
// =================================================================================
// Improved_Gluing_FC_SCL.scl
// Function: FC_Save_Current_Values_V6
// Version: 6.0 (FINAL)
//
// Description:
// FINAL version incorporating all user feedback.
// This function saves a snapshot of all live machine values into the final
// descriptive recipe structure, "UDT_ST10_Recipe_V3".
//
// - IAI axes are correctly mapped to the 3-axis gluing nozzle.
// - V90 axes are correctly mapped to their turntable/jig functions.
// - Does not use loops for positions; every parameter is saved explicitly.
//
// The source DBs ("Gluing_Nozzle_X_DB", "Ring_Table_1_DB", etc.) are placeholders
// and must be replaced with the actual DBs containing the live taught values.
// =================================================================================

FUNCTION "FC_Save_Current_Values_V6" : Void
{ S7_Optimized_Access := 'TRUE' }
VAR_TEMP
   // No loop variables needed
END_VAR

BEGIN
    // =================================================================================
    // 3-AXIS GLUING NOZZLE (IAI Axes)
    // =================================================================================
    "DB_ST10_Recipe".Motion.Gluing_Nozzle_X := "Gluing_Nozzle_X_DB".Live.Positions;
    "DB_ST10_Recipe".Motion.Gluing_Nozzle_Y := "Gluing_Nozzle_Y_DB".Live.Positions;
    "DB_ST10_Recipe".Motion.Gluing_Nozzle_Z := "Gluing_Nozzle_Z_DB".Live.Positions;

    // =================================================================================
    // ROTARY AXES (V90 Servos) - CORRECTED MAPPING
    // =================================================================================

    // --- V90 A1: Ring Turntable 1 ---
    "DB_ST10_Recipe".Motion.Ring_Turntable_Axis_1.Home              := "Ring_Table_1_DB".Live.Positions.Home;
    "DB_ST10_Recipe".Motion.Ring_Turntable_Axis_1.Load_Unload_Pos   := "Ring_Table_1_DB".Live.Positions.Load_Unload_Pos;
    "DB_ST10_Recipe".Motion.Ring_Turntable_Axis_1.Work_Pos_1        := "Ring_Table_1_DB".Live.Positions.Work_Pos_1;
    "DB_ST10_Recipe".Motion.Ring_Turntable_Axis_1.Work_Pos_2        := "Ring_Table_1_DB".Live.Positions.Work_Pos_2;
    // ...etc for spares

    // --- V90 A2: Shaft Scan Turntable ---
    "DB_ST10_Recipe".Motion.Shaft_Scan_Turntable_Axis.Home              := "Shaft_Scan_Table_DB".Live.Positions.Home;
    "DB_ST10_Recipe".Motion.Shaft_Scan_Turntable_Axis.Load_Unload_Pos   := "Shaft_Scan_Table_DB".Live.Positions.Load_Unload_Pos;
    "DB_ST10_Recipe".Motion.Shaft_Scan_Turntable_Axis.Work_Pos_1        := "Shaft_Scan_Table_DB".Live.Positions.Work_Pos_1;
    "DB_ST10_Recipe".Motion.Shaft_Scan_Turntable_Axis.Work_Pos_2        := "Shaft_Scan_Table_DB".Live.Positions.Work_Pos_2;
    // ...etc for spares

    // --- V90 A3: Gluing Rotary Jig ---
    "DB_ST10_Recipe".Motion.Gluing_Rotary_Jig_Axis.Home              := "Gluing_Jig_DB".Live.Positions.Home;
    "DB_ST10_Recipe".Motion.Gluing_Rotary_Jig_Axis.Load_Unload_Pos   := "Gluing_Jig_DB".Live.Positions.Load_Unload_Pos;
    "DB_ST10_Recipe".Motion.Gluing_Rotary_Jig_Axis.Work_Pos_1        := "Gluing_Jig_DB".Live.Positions.Work_Pos_1;
    "DB_ST10_Recipe".Motion.Gluing_Rotary_Jig_Axis.Work_Pos_2        := "Gluing_Jig_DB".Live.Positions.Work_Pos_2;
    // ...etc for spares

    // --- V90 A4: Ring Turntable 2 ---
    "DB_ST10_Recipe".Motion.Ring_Turntable_Axis_2.Home              := "Ring_Table_2_DB".Live.Positions.Home;
    "DB_ST10_Recipe".Motion.Ring_Turntable_Axis_2.Load_Unload_Pos   := "Ring_Table_2_DB".Live.Positions.Load_Unload_Pos;
    "DB_ST10_Recipe".Motion.Ring_Turntable_Axis_2.Work_Pos_1        := "Ring_Table_2_DB".Live.Positions.Work_Pos_1;
    "DB_ST10_Recipe".Motion.Ring_Turntable_Axis_2.Work_Pos_2        := "Ring_Table_2_DB".Live.Positions.Work_Pos_2;
    // ...etc for spares

    // =================================================================================
    // ROBOT GRIPPER FIXTURE CODES
    // =================================================================================

    "DB_ST10_Recipe".Production.Fixtures.Shaft_Handling_Robot.Gripper_A := "Robot1_DB".Live.Gripper_A.FixtureCodes;
    "DB_ST10_Recipe".Production.Fixtures.Shaft_Handling_Robot.Gripper_B := "Robot1_DB".Live.Gripper_B.FixtureCodes;
    "DB_ST10_Recipe".Production.Fixtures.Main_Assembly_Robot.Gripper_A  := "Robot2_DB".Live.Gripper_A.FixtureCodes;
    "DB_ST10_Recipe".Production.Fixtures.Main_Assembly_Robot.Gripper_B  := "Robot2_DB".Live.Gripper_B.FixtureCodes;
    "DB_ST10_Recipe".Production.Fixtures.Unloading_Robot.Gripper_A      := "Robot3_DB".Live.Gripper_A.FixtureCodes;
    "DB_ST10_Recipe".Production.Fixtures.Unloading_Robot.Gripper_B      := "Robot3_DB".Live.Gripper_B.FixtureCodes;

    // =================================================================================
    // OTHER PARAMETERS (Header, Config, Process, etc.)
    // =================================================================================
    "DB_ST10_Recipe".Header.RecipeName       := "System_DB".ActiveRecipe.Name;
    "DB_ST10_Recipe".Header.PartType         := "System_DB".ActivePart.TypeName;
    "DB_ST10_Recipe".Header.RecipeID         := "System_DB".ActiveRecipe.ID;
    "DB_ST10_Recipe".Header.Version          := "System_DB".ActiveRecipe.Version + 1;
    "DB_ST10_Recipe".Header.LastModified     := LTIME_TO_DTL(LTIME());
    "DB_ST10_Recipe".cfg.StationID           := "Station_Config_DB".ID;
    "DB_ST10_Recipe".cfg.PrevStationID       := "Station_Config_DB".Prev_ID;
    "DB_ST10_Recipe".General.StepTimeout     := "Global_Process_Params_DB".Timeouts.Step;
    "DB_ST10_Recipe".General.StepWarning     := "Global_Process_Params_DB".Timeouts.Warning;
    "DB_ST10_Recipe".Process.Limits.RetryLimit := "Global_Process_Params_DB".Limits.Retries;
    "DB_ST10_Recipe".Process.Press.Curve := "Press_B1_Device_DB".ActiveCurve;
    "DB_ST10_Recipe".Process.Press.B1_Program := "Press_B1_Device_DB".ActiveProgram;
    "DB_ST10_Recipe".Process.Press.B2_Program := "Press_B2_Device_DB".ActiveProgram;
    "DB_ST10_Recipe".Process.ATEQ.Pressure_UL := "ATEQ_Device_DB".Limits.Pressure_UL;
    "DB_ST10_Recipe".Process.ATEQ.Pressure_LL := "ATEQ_Device_DB".Limits.Pressure_LL;
    "DB_ST10_Recipe".Process.ATEQ.Leak_UL     := "ATEQ_Device_DB".Limits.Leak_UL;
    "DB_ST10_Recipe".Process.ATEQ.Leak_LL     := "ATEQ_Device_DB".Limits.Leak_LL;
    "DB_ST10_Recipe".Process.ATEQ.PosPressureProgNo := "ATEQ_Device_DB".Programs.Positive;
    "DB_ST10_Recipe".Process.ATEQ.NegPressureProgNo := "ATEQ_Device_DB".Programs.Negative;
    "DB_ST10_Recipe".Process.Timers.Delay_Short      := "Global_Process_Params_DB".Delays.Short;
    "DB_ST10_Recipe".Process.Timers.Delay_Medium     := "Global_Process_Params_DB".Delays.Medium;
    "DB_ST10_Recipe".Process.Timers.Delay_Long       := "Global_Process_Params_DB".Delays.Long;
    "DB_ST10_Recipe".Process.Timers.Cylinder_ActTime := "Global_Process_Params_DB".Delays.Cylinder;
    "DB_ST10_Recipe".Process.Vision.CGlueShaftIV3_Progs := "Vision_System_DB".Shaft_Progs;
    "DB_ST10_Recipe".Process.Vision.CGlueMagnetIV3_Prog  := "Vision_System_DB".Magnet_Prog;
    "DB_ST10_Recipe".Process.Vision.CGlueProgram       := "Vision_System_DB".Glue_Prog;

END_FUNCTION
// NOTE: I used a simplified assignment for the gluing nozzle positions (copying the whole struct).
// If your source DB doesn't match this structure, you will need to expand it
// to assign each position individually, like I did in the V4/V5 functions.
